FUNCTION_BLOCK UDINT_Param
VAR_INPUT PERSISTENT
	val			: UDINT;
END_VAR

END_FUNCTION_BLOCK

(* stored: Version 1.1.0.1
   POU UDINT_Param: Id {aba60908-bb58-49bc-8100-f086aa5743d1}, SpecialFunc None *)
